(* IEC 61131-3 sources: JaccoSigma/tempclass/Class/Class_Names, 1 file *)

(* ---- Class_Names.st ---- *)
(*!
<Class
	Name               = "Class_Names"
	Revision           = "0.0"
	RealtimeTask       = "false"
	CyclicTask         = "false"
	BackgroundTask     = "false"
	Sigmatek           = "false"
	OSInterface        = "false"
	HighPriority       = "false"
	Automatic          = "false"
	UpdateMode         = "Prescan"
	SharedCommandTable = "true"
	Objectsize         = "(484,120)">
	<Channels>
		<Server Name="Client_Counter" Visualized="false" Initialize="false" WriteProtected="true" Retentive="false"/>
		<Server Name="Server0" Visualized="false" Initialize="false" WriteProtected="true" Retentive="false"/>
		<Server Name="Server1" Visualized="false" Initialize="false" WriteProtected="true" Retentive="false"/>
		<Server Name="Server_Counter" Visualized="false" Initialize="false" WriteProtected="true" Retentive="false"/>
		<Client Name="_SigCLib" Required="false" Internal="false"/>
		<Client Name="Client" Required="false" Internal="false"/>
		<Client Name="Client0" Required="false" Internal="false"/>
		<Client Name="Client1" Required="false" Internal="false"/>
		<Client Name="Client2" Required="false" Internal="false"/>
	</Channels>
</Class>
*)
Class_Names : CLASS
	TYPE
	  Names : ARRAY [0..100] OF CHAR;  //! <Type Public="true" Name="Names"/>
	END_TYPE
  //Servers:
	Server_Counter 	: SvrChCmd_DINT;
	Client_Counter 	: SvrCh_DINT;
	Server0 	: SvrCh_DINT;
	Server1 	: SvrCh_DINT;
  //Clients:
	_SigCLib 	: CltChCmd_SigCLib;
	Client 	: CltChCmd__MultiTask;
	Client0 	: CltCh_DINT;
	Client1 	: CltCh_DINT;
	Client2 	: CltCh_DINT;
  //Variables:
		ServerNames : ARRAY [0..100] OF Names;

		ClientNames : ARRAY [0..100] OF Names;

		ClassName : ARRAY [0..100] OF CHAR;

		ObjectName : ARRAY [0..100] OF CHAR;

		SVRTypes : ARRAY [0..100] OF ChMode;

		CLITypes : ARRAY [0..100] OF ChMode;

		TotalDsc : ARRAY [0..5] OF ChDscEntry;

		first 	: DINT;
  //Functions:

	FUNCTION VIRTUAL GLOBAL Init;

	FUNCTION GLOBAL FindNames;
  //Tables:
	FUNCTION @STD
		VAR_OUTPUT
			ret_code	: CONFSTATES;
		END_VAR;
	FUNCTION GLOBAL TAB @CT_;
END_CLASS;

#pragma usingLtd _MultiTask
#pragma usingLtd SigCLib

FUNCTION VIRTUAL GLOBAL Class_Names::Init
VAR
	ObjectNameSize : UDINT;
  ClassNameSize  : UDINT;
END_VAR

  if _FirstScan = TRUE then
    FindNames();
    ObjectNameSize := _strlen(src:=sigclib_nameof_object(pthis:=this));
    ClassNameSize  := _strlen(src:=sigclib_nameof_class(pthis:=this));
    if sizeof(ObjectName) >= ObjectNameSize & sizeof(ClassName) >= ClassNameSize then
      _strcpy(dest:=#ObjectName[0], src:=sigclib_nameof_object(pthis:=this));
      _strcpy(dest:=#ClassName[0], src:=sigclib_nameof_class(pthis:=this));
    end_if;
  end_if;

END_FUNCTION

FUNCTION GLOBAL Class_Names::FindNames
VAR
  pObject         :^obj;
  pClassHeader    :^ClsHdr;
  IDX             :dint;
  Length          :udint;
  pName           :^char;
  ptype           :^ChMode;
  pTotal          :^ChDscEntry;
END_VAR

  //Pointer to obj header
  pObject           := LSL_GetHdr(this);

  //pointer to class header
  pClassHeader      := pObject^.pClsHdr;
  Server_Counter    := pClassHeader^.pDsc^.nSvrChs;
  Client_Counter    := pClassHeader^.pDsc^.nCltChs;

  pName := #pClassHeader^.aDscChs[0].pDsc^.Name.Text$char;
  ptype := #pClassHeader^.aDscChs[0].pDsc^.uiMode;
  pTotal:= #pClassHeader^.aDscChs[0].pDsc^;

  Length := 0;

  for IDX := 0 to Server_Counter - 1 do //Write all Server names to var
    _strcpy(#ServerNames[IDX][0],pName);
    Length := _strlen(src:=#ServerNames[IDX][0]);
    pName  += (Length+11);

    SVRTypes[IDX] := ptype^;
    ptype += (Length+11);
  end_for;

  for IDX := 0 to Client_Counter - 1 do //Write all Client names to var
    _strcpy(#ClientNames[IDX][0],pName);
    Length := _strlen(src:=#ClientNames[IDX][0]);
    if first < 2 then
      pName  += (Length+27);
      first += 1;
    else
      pName  += (Length+11);
    end_if;

    CLITypes[IDX] := ptype^;
    ptype += (35);

    TotalDsc[idx] := pTotal^;
    pTotal += (32); //length + 11 and "ClassSvr" + 11? lol no luck.
  end_for;

END_FUNCTION
